// TIA Portal V16 export
// export: Created 2022-09-01T14:27:01.9278772Z, ExportSetting WithDefaults, DisplayName Totally Integrated Automation Portal, DisplayVersion V16, DisplayName TIA Portal Version Control Interface, DisplayVersion V16, DisplayName TIA Portal Openness, DisplayVersion V16, DisplayName STEP 7 Professional, DisplayVersion V16, DisplayName STEP 7 Safety, DisplayVersion V16, DisplayName WinCC Advanced, DisplayVersion V16
FUNCTION "Totalizador_Bombas" : Void   // FC10, LAD
{ S7_Optimized_Access := 'TRUE' }
VERSION : 0.1
// stored: AutoNumber true, IsIECCheckEnabled false, SetENOAutomatically false, UDAEnableTagReadback false
BEGIN

REGION Network 1
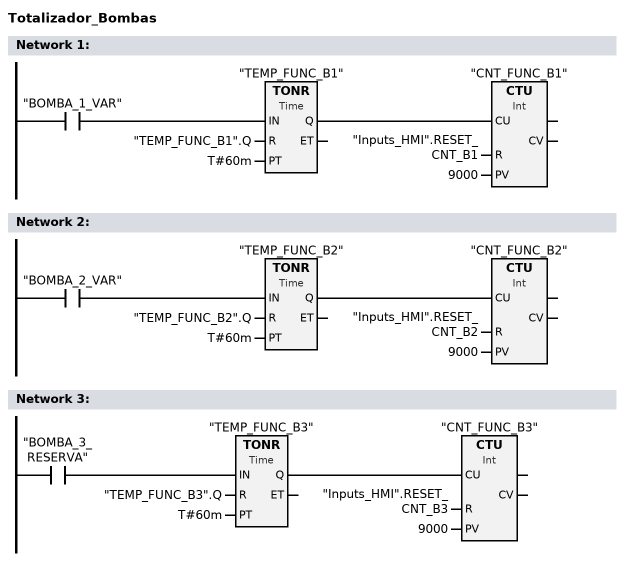
   RUNG wire#powerrail
      Contact( "BOMBA_1_VAR" )
      { S7_Templates := "time_type := Time" } "TEMP_FUNC_B1".TONR(r := "TEMP_FUNC_B1".Q, pt := T#60m, et =>)
      { S7_Templates := "value_type := Int" } "CNT_FUNC_B1".CTU(r := "Inputs_HMI".RESET_CNT_B1, pv := 9000, cv =>)
   END_RUNG
   // the same network as SCL:
   "TEMP_FUNC_B1".TONR(IN := "BOMBA_1_VAR", R := "TEMP_FUNC_B1".Q, PT := T#60m);
   "CNT_FUNC_B1".CTU(CU := "TEMP_FUNC_B1".Q, R := "Inputs_HMI".RESET_CNT_B1, PV := 9000);
END_REGION

REGION Network 2
   RUNG wire#powerrail
      Contact( "BOMBA_2_VAR" )
      { S7_Templates := "time_type := Time" } "TEMP_FUNC_B2".TONR(r := "TEMP_FUNC_B2".Q, pt := T#60m, et =>)
      { S7_Templates := "value_type := Int" } "CNT_FUNC_B2".CTU(r := "Inputs_HMI".RESET_CNT_B2, pv := 9000, cv =>)
   END_RUNG
   // the same network as SCL:
   "TEMP_FUNC_B2".TONR(IN := "BOMBA_2_VAR", R := "TEMP_FUNC_B2".Q, PT := T#60m);
   "CNT_FUNC_B2".CTU(CU := "TEMP_FUNC_B2".Q, R := "Inputs_HMI".RESET_CNT_B2, PV := 9000);
END_REGION

REGION Network 3
   RUNG wire#powerrail
      Contact( "BOMBA_3_RESERVA" )
      { S7_Templates := "time_type := Time" } "TEMP_FUNC_B3".TONR(r := "TEMP_FUNC_B3".Q, pt := T#60m, et =>)
      { S7_Templates := "value_type := Int" } "CNT_FUNC_B3".CTU(r := "Inputs_HMI".RESET_CNT_B3, pv := 9000, cv =>)
   END_RUNG
   // the same network as SCL:
   "TEMP_FUNC_B3".TONR(IN := "BOMBA_3_RESERVA", R := "TEMP_FUNC_B3".Q, PT := T#60m);
   "CNT_FUNC_B3".CTU(CU := "TEMP_FUNC_B3".Q, R := "Inputs_HMI".RESET_CNT_B3, PV := 9000);
END_REGION
END_FUNCTION
